FUNCTION_BLOCK logiBUS_AI_IDA (* Composite FB for analog double word input data *)
  (* Standard: 61499-2; Description: Copyright (c) 2026 HR Agrartechnik GmbH This program and the accompanying materials are made available under the terms of the Eclipse Public License 2.0 which is available at https://www.eclipse.org/legal/epl-2.0/ SPDX-License-Identifier: EPL-2.0 AnalogInput_hysteresis = 0 switches the change trigger off (use 1 to see every change). TimeDelta = 0 or 16#FFFFFFFF switches the cyclic IND off. With both off the block sends no IND (value only via REQ). IN = 0-4095 (12 bit, fixed full-scale raw value, ESP32-P4 ADC continuous/DMA mode has no other bit width to choose from). *)
  (* Version 1.0, 2026-02-23, Franz Höpfinger, HR Agrartechnik GmbH *)
  PACKAGE logiBUS::io::AI;
  IMPORT logiBUS::io::AI::logiBUS_AI::Invalid;
  (* Documentation:
  logiBUS_AI_IDA
   🇩🇪 Deutsch
   Composite-Baustein, der den Service-Interface-Baustein logiBUS_AI_ID um eine Adapter-Schnittstelle erweitert: Der Rohwert steht statt über die klassischen IN/CNF/IND-Ereignisse als Plug IN (Typ adapter::types::unidirectional::AD) bereit, zusätzlich kann über den Socket SREQ ein externer Adapter eine Abfrage anstoßen (per E_R_TRIG flankengetriggert auf REQ).
   Schnittstelle
    - INIT (mit QI, PARAMS, Input, AnalogInput_hysteresis, TimeDelta, TimeRateLimit): wie logiBUS_AI_ID, wird direkt durchgereicht.
   - REQ (mit QI): sofortige Abfrage; kann zusätzlich über den Socket SREQ extern ausgelöst werden.
   - INITO (mit QO, STATUS): Bestätigung der Initialisierung.
   - Plug IN (adapter::types::unidirectional::AD): liefert den Rohwert als Adapter-Ereignis/-Daten (E1/D1) statt der einzelnen CNF/IND-Events des inneren Bausteins.
   - Socket SREQ (adapter::types::unidirectional::AX): externe Service-Anforderung, über E_R_TRIG flankengetriggert auf AI.REQ.
    Roh-Vollausschlag von IN
   Wie beim inneren Baustein logiBUS_AI_ID: IN liefert den ADC-Rohwert im Bereich 0-4095 (12 bit), auf dem ESP32-P4 im Continuous/DMA-ADC-Modus fix (keine andere Bit-Breite wählbar). Details und Umrechnung Rohwert→Volt siehe dort.
   🇬🇧 English
   Composite block that extends the service interface block logiBUS_AI_ID with an adapter interface: instead of the classic IN/CNF/IND events, the raw value is exposed as a plug IN (type adapter::types::unidirectional::AD); additionally, an external adapter can trigger a read via the socket SREQ (edge-triggered onto REQ via E_R_TRIG).
   Interface
    - INIT (with QI, PARAMS, Input, AnalogInput_hysteresis, TimeDelta, TimeRateLimit): same as logiBUS_AI_ID, passed straight through.
   - REQ (with QI): immediate read; can also be triggered externally via the SREQ socket.
   - INITO (with QO, STATUS): initialization confirmation.
   - Plug IN (adapter::types::unidirectional::AD): delivers the raw value as an adapter event/data pair (E1/D1) instead of the internal block's individual CNF/IND events.
   - Socket SREQ (adapter::types::unidirectional::AX): external service request, edge-triggered onto AI.REQ via E_R_TRIG.
    Raw full-scale value of IN
   Same as the internal logiBUS_AI_ID block: IN delivers the raw ADC value in the range 0-4095 (12 bit), fixed on the ESP32-P4 in continuous/DMA ADC mode (no other bit width selectable). See there for details and the raw-to-volt conversion.
  *)
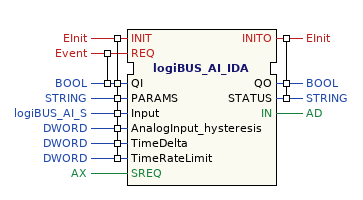
  EVENT_INPUT
    INIT : EInit WITH QI, PARAMS, Input, AnalogInput_hysteresis, TimeDelta, TimeRateLimit; (* Service Initialization *)
    REQ WITH QI; (* Service Request *)
  END_EVENT
  EVENT_OUTPUT
    INITO : EInit WITH QO, STATUS; (* Initialization Confirm *)
  END_EVENT
  VAR_INPUT
    QI : BOOL; (* Event Input Qualifier *)
    PARAMS : STRING; (* Service Parameters *)
    Input : logiBUS::io::AI::logiBUS_AI_S := Invalid; (* Identify the Input Input_I1..I8 *)
    AnalogInput_hysteresis : DWORD; (* IND when the raw value changes by more than this (0 = off) *)
    TimeDelta : DWORD := 250; (* After How many ms an IND (poll interval, 0 or 16#FFFFFFFF = off) *)
    TimeRateLimit : DWORD := 100; (* Maximum 1 IND in how many ms. (< delta) *)
  END_VAR
  VAR_OUTPUT
    QO : BOOL; (* Event Output Qualifier *)
    STATUS : STRING; (* Service Status *)
  END_VAR
  SOCKETS
    SREQ : adapter::types::unidirectional::AX; (* Service Request *)
  END_SOCKETS
  PLUGS
    IN : adapter::types::unidirectional::AD; (* Input data from resource, raw value 0-4095 (12 bit, fixed ESP32-P4 ADC continuous-mode full scale) *)
  END_PLUGS
  FBS
    AI : logiBUS::io::AI::logiBUS_AI_ID;
    E_R_TRIG : iec61499::events::E_R_TRIG;
  END_FBS
  EVENT_CONNECTIONS
    INIT TO AI.INIT;
    AI.INITO TO INITO;
    AI.IND TO IN.E1;
    AI.CNF TO IN.E1;
    REQ TO AI.REQ;
    E_R_TRIG.EO TO AI.REQ;
    SREQ.E1 TO E_R_TRIG.EI;
  END_CONNECTIONS
  DATA_CONNECTIONS
    AI.IN TO IN.D1;
    QI TO AI.QI;
    PARAMS TO AI.PARAMS;
    AI.QO TO QO;
    AI.STATUS TO STATUS;
    Input TO AI.Input;
    AnalogInput_hysteresis TO AI.AnalogInput_hysteresis;
    SREQ.D1 TO E_R_TRIG.QI;
    TimeDelta TO AI.TimeDelta;
    TimeRateLimit TO AI.TimeRateLimit;
  END_CONNECTIONS
END_FUNCTION_BLOCK
